// TIA Portal V18 export
// export: Created 2026-03-12T16:04:34.7684012Z, ExportSetting WithDefaults, DisplayName Totally Integrated Automation Portal, DisplayVersion V18 Update 5, DisplayName TIA Portal Openness, DisplayVersion V18 Update 5, DisplayName TIA Portal Version Control Interface, DisplayVersion V18, DisplayName SINAMICS Startdrive Advanced, DisplayVersion V18, DisplayName SINAMICS Startdrive G130, G150, S120, S150, SINAMICS MV, S210, DisplayVersion V18, DisplayName SINAMICS Startdrive G110M, G120, G120C, G120D, G120P, G115D, DisplayVersion V18, DisplayName STEP 7 Professional, DisplayVersion V18 Update 5, DisplayName STEP 7 Safety, DisplayVersion V18, DisplayName WinCC Professional, DisplayVersion V18 Update 5
FUNCTION_BLOCK "FB_HORÍMETRO"   // FB22, LAD
TITLE = Function Block HORÍMETRO - Contador de Horas
{ S7_Optimized_Access := 'TRUE' }
VERSION : 0.1
// Bloco para realizar a contagem de quantas horas cada motor/bomba passou ligado.
// stored: AutoNumber true, IsIECCheckEnabled false, IsRetainMemResEnabled false, MemoryReserve 100, SetENOAutomatically false, UDAEnableTagReadback false
   VAR_INPUT
      INPUT_LIGADO : Bool;   // Entrada do sinal de falha instanciado na Network 1
      INPUT_RESET_HORIMETRO : Bool;   // Entrada do sinal de reset horímetro (horas trabalhadas da bomba)
   END_VAR
   VAR_IN_OUT
      HORIMETRO : UInt;   // Saída do horímetro (horas trabalhadas da bomba)
   END_VAR
   VAR RETAIN
      RESET_SEGUNDO : Bool;   // Comando para zerar as horas acumuladas
      MINUTO : Bool;   // Pulso para contador de minutos
      COUNT_MINUTO : Bool;   // Contador de minutos
      RESET_MINUTO : Bool;   // Reset do contador de minutos
      HORA : Bool;   // Pulso para contador de horas
      COUNT_HORA : Bool;   // Contador de horas
      HORAS : UInt;   // Horas armazenadas para mover ao Horimetro e zerar quando solicitado
      TIMER_SEGUNDO : IEC_COUNTER;   // Bloco contador de segundos
      TIMER_MINUTO : IEC_COUNTER;   // Bloco contador de minutos
   END_VAR
BEGIN

REGION Network 1: Acumulação de horas (Utilizando clock de 1Hz/1s)
   // TIMER_SEGUNDO: Bloco contador de segundos
   // TIMER_MINUTO: Bloco contador de minutos
   // INC: Incremento de horas
   // RESET_HORIMETRO: Comando para zerar as horas acumuladas
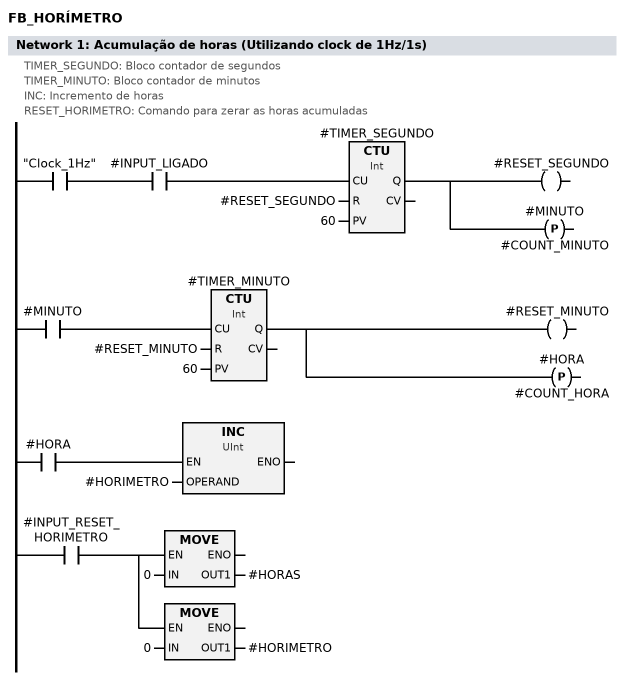
   #TIMER_SEGUNDO.CTU(CU := "Clock_1Hz" AND #INPUT_LIGADO, R := #RESET_SEGUNDO, PV := 60);
   #RESET_SEGUNDO := #TIMER_SEGUNDO.Q;
   #MINUTO := #TIMER_SEGUNDO.Q AND NOT #COUNT_MINUTO;   // rising edge
   #COUNT_MINUTO := #TIMER_SEGUNDO.Q;
   #TIMER_MINUTO.CTU(CU := #MINUTO, R := #RESET_MINUTO, PV := 60);
   #RESET_MINUTO := #TIMER_MINUTO.Q;
   #HORA := #TIMER_MINUTO.Q AND NOT #COUNT_HORA;   // rising edge
   #COUNT_HORA := #TIMER_MINUTO.Q;
   IF #HORA THEN #HORIMETRO := #HORIMETRO + 1; END_IF;
   IF #INPUT_RESET_HORIMETRO THEN
       #HORAS := 0;
       #HORIMETRO := 0;
   END_IF;
END_REGION
END_FUNCTION_BLOCK
